{attribute 'hide_all_locals' := ''}
{attribute 'FBVisuCreator' := ''}
{attribute 'FBVisuCreatorPrefix' := 'RET_VISU_'}
FUNCTION_BLOCK Strecke
VAR_INPUT
	{attribute 'FBVisuCreatorFormatString' := '%1.3f'}
	fX: REAL;
	{attribute 'FBVisuCreatorFormatString' := '%1.3f'}
	fRauschen: REAL;
	{attribute 'FBVisuCreatorFormatString' := '%1.3f'}
	fOffset: REAL;
	{attribute 'FBVisuCreatorBoolColor' := 'Green'}
	bNichtlinear: BOOL;
END_VAR
VAR_OUTPUT
	{attribute 'FBVisuCreatorFormatString' := '%1.3f'}
	fY: REAL;
END_VAR
VAR
	{attribute 'hide'}
	fbLinearisierung: Kennlinie := (bAktiviert := TRUE, bSpiegelungXgY := FALSE, fXin_0 := 0.0, fXin_1 := 10.0, fXin_2 := 20.0, fXin_3 := 30.0, fXin_4 := 40.0, fXin_5 := 50.0, fXin_6 := 60.0, fXin_7 := 70.0, fXin_8 := 80.0, fXin_9 := 90.0, fXin_10 := 100.0, fYin_0 := 0.0, fYin_1 := 2.5, fYin_2 := 5.0, fYin_3 := 12.5, fYin_4 := 20.0, fYin_5 := 30.0, fYin_6 := 40.0, fYin_7 := 47.5, fYin_8 := 65.0, fYin_9 := 77.5, fYin_10 := 90.0);
	{attribute 'hide'}
	fbPT1: PT1 := (fK := 0.75, fT := 0.5);
	{attribute 'hide'}
	fbRauschen: Rauschen := (fVerstaerkung := 0.0);
END_VAR
VAR // added by the converter: edge detectors and wires of the graphical bodies
    _w1 : ANY;
    _w2 : REAL;
END_VAR

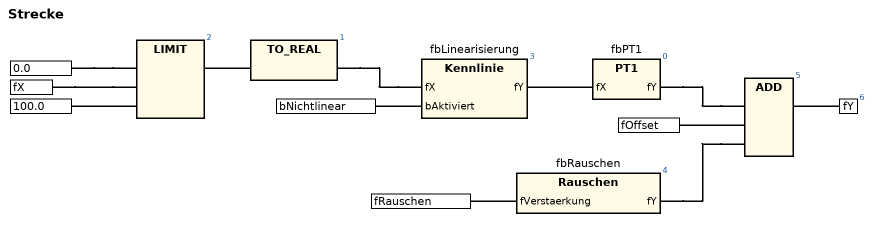
fbPT1(fX := fbLinearisierung.fY); // PT1
_w2 := TO_REAL(_w1);
_w1 := LIMIT(0.0, fX, 100.0);
fbLinearisierung(fX := _w2, bAktiviert := bNichtlinear); // Kennlinie
fbRauschen(fVerstaerkung := fRauschen); // Rauschen
fY := fbPT1.fY + fOffset + fbRauschen.fY;

END_FUNCTION_BLOCK

(* stored: Version 1.1.0.1, ProductVersion 3.1.4024.12
   POU Strecke: Id {9b79c57c-432a-4b8c-b851-e17d31b48f66}, SpecialFunc None *)
